TYPE ST_DebugSensors_TurnTableDtuEmulation :
STRUCT
	EnableSensorDebug	: BOOL; 					// Overwrite sensor values with debug sensor values
	HW_Inputs			: ST_HW_InputsTurnTableDTU;	// Debug sensors
END_STRUCT
END_TYPE

(* stored: Version 1.1.0.1, ProductVersion 3.1.4024.9
   DUT ST_DebugSensors_TurnTableDtuEmulation: Id {00b65960-a162-4348-ab30-1268caa4764d} *)
